Staubli VAL3: MotionCfgVel.dtx

public frame fReference = {fatherId=world[0]}
public mdesc mMaxSpeed
public tool tTool = {fatherId=flange[0], ioLink=valve1}
public num nCmdType
